{attribute 'qualified_only'}
{attribute 'strict'}
TYPE mqttExtraCode :
(
	sendNothing := 0,
	sendIdle,
	sendCharging1,
	sendCharging2	
);
END_TYPE

(* stored: Version 1.1.0.1, ProductVersion 3.1.4024.11
   DUT mqttExtraCode: Id {7e43c804-74c8-4d74-a264-f94da94da31b} *)
